TYPE TFPortaStatus :
STRUCT
	PortaAperta 	: BOOL;
	PortaChiusa 	: BOOL;
	AnomaliaPorta 	: BOOL;
END_STRUCT
END_TYPE

(* stored: Version 1.1.0.1, ProductVersion 3.1.4024.11
   DUT TFPortaStatus: Id {d36961ea-093e-4443-82c9-0a6418f143d6} *)
